FUNCTION_BLOCK ZONA6 EXTENDS ZONA

VAR_INPUT
	i3		:	BOOL;
	i9		:	BOOL;
END_VAR

VAR_OUTPUT
	q10		:	BOOL;
END_VAR

VAR
	Tdelay1	:	TOF();
	Tdelay	:	TON();
	stato: ( S0, S1, S2, S3) := S0;
END_VAR

 IF ENABLE = FALSE THEN
	 stato := S0;
 END_IF


 CASE stato OF 

	 S0:
	 q10 := FALSE;
	 IF i3 = FALSE AND i9 = FALSE THEN
		 stato := S1;
	 END_IF
	 
	 S1:
	 Tdelay ( IN := stato = S1, PT := T#500MS);
	 IF Tdelay.Q = TRUE THEN
		 stato := S2;
	 END_IF
	 
	 S2:
	 q10 := TRUE;
	 IF i9 = TRUE THEN
		 stato := S3;
	 END_IF
	 
	 S3:
	 Tdelay1 ( IN := (stato = S3), PT := T#500MS);
	 IF Tdelay.Q = TRUE THEN
		 stato := S0;
	 END_IF
	 
 END_CASE

END_FUNCTION_BLOCK

(* stored: Version 1.1.0.1, ProductVersion 3.1.4024.12
   POU ZONA6: Id {c84eebd9-b60a-4fa5-9768-5cd1c72271a9}, SpecialFunc None *)
